(* CoDeSys 2.3 export: LogDint.EXP *)

(* POU basic/LogDint, ST *)
FUNCTION LogDint : BOOL
VAR_INPUT
    Value: DINT;
    Channel: UINT;
END_VAR
VAR
END_VAR
IF Channel < 256 THEN
    EvtCh8Tick32Int32(UINT_TO_BYTE(Channel), GlobalTick, Value, GlobalLogBufferHandle);
ELSE
    EvtCh16Tick32Int32(Channel, GlobalTick, Value, GlobalLogBufferHandle);
END_IF
END_FUNCTION
